FUNCTION_BLOCK AOI_CountersAdmin
VAR_INPUT
	Enable: BOOL; //启用
	Execute: BOOL; //数粒信号
	Reset: bool; //重置
    In_Total: DINT; //计划生产总数
	Quantity: DINT;
	Clear: BOOL;//清除故障
	SkipAlarm: BOOL;
	CheckTime: DINT;
    CheckCnt: BOOL;
	ManualCnt: BOOL;
END_VAR
VAR_OUTPUT
	DropVibrator_Wrk: BOOL;//落料启动
	CircleVibrator_Wrk: BOOL;//圆震启动
	LineVibrator_Wrk: BOOL;//直震启动
	Warning: BOOL;	
	Busy: BOOL;//数粒中
	Error: BOOL; //报警
	ErrorID: DINT;//报警代码;	
	InitDone: BOOL;//初始化完成
	Out_Total: DINT;//实际生产数量
	Complete: BOOL; //生产完成
	CntUp: DINT;
	ProcessTime : DINT;//
	Speed: REAL;
	_diLastCnt: ARRAY[0..100] OF DINT;
END_VAR
VAR
	iAxisAct: INT;	
	tonHighCheck: TON;
	tonLowCheck: TON;
	tonLackCheck: TON;
	tonWatchDog: TON;
	tonProcess: TON;
	tonEnable: TON;
	rt_Exe: R_TRIG;	
	aoi_DropSensor: AOI_Sensoradmin;
	aoi_LowSensor: AOI_Sensoradmin;
	aoi_HighSensor: AOI_Sensoradmin;	
	lrPosAdd: LREAL;
	rt_Clear: R_TRIG; 
	rt_Drop: R_TRIG;
	rtLowCheck: R_trig;
	toncheck: TON;
	diLastTargetCnt: DINT;
	QuantityBuffer: DINT;
	tonDropDelay: Ton;
	diCheckFaultCnt: DINT;
	diFaultCnt: ARRAY[0..64] OF dint;
	i: INT;
	CntLost: DINT;
	
	rtFaultcnt: R_trig;
END_VAR
VAR_IN_OUT
	Axis: UDT_AxisAdmin;//数粒伺服
	DropSensor: UDT_SensorAdmin;//缺料检测
	LowSensor: UDT_SensorAdmin;//低料位检测
	HighSensor: UDT_SensorAdmin;//高料位检测
	Cylinder: UDT_CylinderAdmin;//
	DropFlag: BOOL;//
END_VAR

rt_Exe(CLK:=Execute , Q=> );
rt_Drop(CLK:= DropSensor.o.Value, Q=> );
tonEnable(IN:= Enable, PT:= T#3S, Q=> , ET=> );
IF NOT Enable THEN		
	DropVibrator_Wrk:=FALSE;//震动盘启动
	CircleVibrator_Wrk:=FALSE;
	LineVibrator_Wrk:=FALSE;	
END_IF

IF Enable THEN
   IF NOT HighSensor.o.Value  AND NOT Complete THEN
	  DropVibrator_Wrk:=TRUE;//落料震动盘启动
	  ELSE
	  DropVibrator_Wrk:=FALSE;//
   END_IF
   IF NOT LowSensor.o.Value AND NOT Complete  THEN	  
	   CircleVibrator_Wrk:=TRUE;//圆震动盘启动
	   ELSE
	   CircleVibrator_Wrk:=FALSE;	   
   END_IF	
   CircleVibrator_Wrk:= TRUE;
   LineVibrator_Wrk:= TRUE;//直震动盘启动常开
ELSE
   DropVibrator_Wrk:=FALSE;
   LineVibrator_Wrk:= FALSE;
   CircleVibrator_Wrk:= FALSE;
END_IF

IF reset THEN
	Complete:=FALSE;
	Out_Total:=0;
END_IF

rt_Clear(CLK:= Clear, Q=> );
IF rt_Clear.Q THEN
   Error:=FALSE;
END_IF

IF Enable AND Quantity=0 THEN
	IF DropFlag THEN
	   DropFlag:=FALSE;
	END_IF
END_IF

CASE iAxisAct OF
	0: 
        Busy:=FALSE;
		IF Out_Total<In_Total AND Quantity<>0 AND tonEnable.Q THEN
		   QuantityBuffer:=Quantity;
		   iAxisAct:=10;
		ELSE IF Out_Total=In_Total THEN
				Complete:=TRUE;
		     END_IF
		END_IF

	10:
	    IF QuantityBuffer>20 THEN
		   QuantityBuffer:=QuantityBuffer-20;
		   iAxisAct:=11;
		ELSE
           iAxisAct:=12;   
	    END_IF
	   
	11:
	    Busy:=TRUE;
		CntUp:=0;
	    lrPosAdd:=20*360/24; 
		diLastTargetCnt:=20;
	    Axis.i.Pos:=lrPosAdd;
		iAxisAct:=20;
		
	12: 
	    Busy:=TRUE;
		CntUp:=0;
	    lrPosAdd:=QuantityBuffer*360/24; 
		diLastTargetCnt:=QuantityBuffer;
		QuantityBuffer:=0;
	    Axis.i.Pos:=lrPosAdd;
		iAxisAct:=20;
	    
	20:
	    Axis.i.MoveAdd:=TRUE;
	    tonProcess(IN:=TRUE , PT:=T#100S , Q=> , ET=> );
	    ProcessTime:= TIME_TO_DINT(tonProcess.ET);
		IF Axis.o.CmdDone OR Axis.o.Error THEN
		   Axis.i.MoveAdd:=FALSE;
		   iAxisAct:=30;
		   tonProcess(IN:=FALSE , PT:=T#100S , Q=> , ET=> );
		   Speed:=1000/DINT_TO_REAL(ProcessTime);
		END_IF
	30:

		toncheck(IN:= TRUE, PT:= DINT_TO_TIME(CheckTime), Q=> , ET=> );
		
	    IF NOT SkipAlarm AND toncheck.Q AND CntUp<1  THEN
		   Error:=TRUE;
		END_IF
(*		
		IF NOT CheckCnt AND toncheck.Q AND CntUp <> diLastTargetCnt THEN
		   Error:=TRUE;
		END_IF	
	
        rtFaultcnt(CLK:= toncheck.Q  , Q=> );
		IF toncheck.Q  THEN
			
		   diFaultCnt[i]:= diLastTargetCnt - CntUp;
		   _diLastCnt[i]:= CntUp;
		   i:=i+1;
		   IF i>60 THEN
			   i:=0;
		   END_IF
		    
		END_IF
		
		
		IF (SkipAlarm AND CheckCnt)OR toncheck.Q THEN
		   toncheck(IN:= FALSE, PT:= DINT_TO_TIME(CheckTime), Q=> , ET=> );
           iAxisAct:=100;
		END_IF
*)
//20221206		
        
		IF (SkipAlarm AND CheckCnt)OR 
            toncheck.Q THEN
			
		    toncheck(IN:= FALSE, PT:= DINT_TO_TIME(CheckTime), Q=> , ET=> );	
			CntLost:=diLastTargetCnt-CntUp;
			
			
		   diFaultCnt[i]:= CntLost;
		   _diLastCnt[i]:= CntUp;
		   i:=i+1;
		   IF i>60 THEN
			   i:=0;
		   END_IF		
			

			IF CntLost>0 THEN
		       iAxisAct:=40;
			ELSE
               iAxisAct:=100;
			END_IF
			
		END_IF	
		
	40:		
	    diCheckFaultCnt:=diCheckFaultCnt+1;
		CntUp:=0;
	    lrPosAdd:=CntLost*360/24;
	    Axis.i.Pos:=lrPosAdd;
		iAxisAct:=41;		
		
	41:
		
	    Axis.i.MoveAdd:=TRUE;
		IF Axis.o.CmdDone OR Axis.o.Error THEN
		   Axis.i.MoveAdd:=FALSE;
		   iAxisAct:=42;
		END_IF
	
	42:
	
		toncheck(IN:= TRUE, PT:= DINT_TO_TIME(CheckTime), Q=> , ET=> );
		
		IF NOT CheckCnt AND toncheck.Q AND CntUp <> CntLost THEN
		   Error:=TRUE;
		END_IF	
		
		IF (SkipAlarm AND CheckCnt)OR toncheck.Q THEN
		   toncheck(IN:= FALSE, PT:= DINT_TO_TIME(CheckTime), Q=> , ET=> );
		   CntLost:=0;
           iAxisAct:=100;
		END_IF		
		
		
		
		
	100:	
	    Busy:=FALSE;
		IF NOT Cylinder.i.OutSensor AND NOT Cylinder.i.InSensor THEN
		   Cylinder.i.ActiveIn:=TRUE;
		   Cylinder.i.ActiveOut:=FALSE;
		END_IF
		
		IF DropFlag AND NOT Error THEN
		   IF Cylinder.i.OutSensor THEN
		      iAxisAct:=110;
           END_IF	
		   IF Cylinder.i.InSensor THEN
		      iAxisAct:=120;
           END_IF	
		END_IF		
		IF Error AND rt_Drop.Q THEN
		   iAxisAct:=101;
		END_IF
		
		IF Reset THEN
		   iAxisAct:=0;
        END_IF
		
	101:	
		Axis.i.Pos:=360/24;
	    Axis.i.MoveAdd:=TRUE;
		IF Axis.o.CmdDone OR Axis.o.Error THEN
		   Axis.i.MoveAdd:=FALSE;
		   iAxisAct:=102;
		END_IF		
	102:
	    tonDropDelay(IN:= TRUE, PT:= T#1S, Q=> , ET=> );
		IF tonDropDelay.Q THEN
			tonDropDelay(IN:= FALSE, PT:= T#1S, Q=> , ET=> );
			iAxisAct:=100;
		END_IF
		
	110: 
	    Cylinder.i.ActiveIn:=TRUE;
		Cylinder.i.ActiveOut:=FALSE;
		IF Cylinder.i.InSensor THEN
			iAxisAct:=200;
		END_IF
		
	120:
	    Cylinder.i.ActiveIn:=FALSE;
		Cylinder.i.ActiveOut:=TRUE;
		IF Cylinder.i.OutSensor THEN
			iAxisAct:=200;
		END_IF	
	200:
	    IF QuantityBuffer=0 THEN
		   iAxisAct:=300;
		ELSE 
		   iAxisAct:=10;
		END_IF
	
	300:
	    Out_Total:=Out_Total+1; 
        DropFlag:=FALSE;
	    iAxisAct:=0;
	
END_CASE

tonHighCheck(IN:= NOT HighSensor.o.Value AND Enable AND Quantity<>0 , PT:=T#15S , Q=> , ET=> );
tonLowCheck(IN:= NOT LowSensor.o.Value  AND Enable, PT:=T#5S , Q=> , ET=> );
rtLowCheck(CLK:= LowSensor.o.Value, Q=> );

IF rtLowCheck.Q THEN
   CntUp:=CntUp+1;
END_IF

Warning:= tonHighCheck.Q AND NOT Error ;

aoi_DropSensor(Admin:= DropSensor);
aoi_HighSensor(Admin:= HighSensor);
aoi_LowSensor(Admin:= LowSensor);

(*
 rtFaultcnt(CLK:=   , Q=> );
IF rtFaultcnt.Q THEN
	MEMSET(destAddr:= ADR(diFaultCnt), fillByte:= 0, n:=SIZEOF(diFaultCnt) );
	MEMSET(destAddr:= ADR(_diLastCnt), fillByte:= 0, n:=SIZEOF(_diLastCnt) );
END_IF
*)

END_FUNCTION_BLOCK

(* stored: Version 1.1.0.1, ProductVersion 3.1.4024.6
   POU AOI_CountersAdmin: Id {c9f10a5c-022c-49bf-bdab-f98c0a987401}, SpecialFunc None *)
